SUBAPPLICATION mapping_Uebung_010b3 (* Toggle Flip-Flop mit IE AuxFunction2_X1 *)
  (* Standard: 61499-2; Description: Copyright (c) 2023 Meisterschulen am Ostbahnhof This program and the accompanying materials are made available under the terms of the Eclipse Public License 2.0 which is available at https://www.eclipse.org/legal/epl-2.0/ SPDX-License-Identifier: EPL-2.0 *)
  (* Version 1.0, 2023-10-23, Franz Höpfinger, Meisterschulen am Ostbahnhof *)
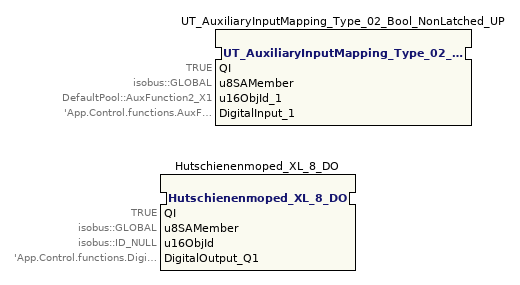
  FBS
    Hutschienenmoped_XL_8_DO : Hutschienenmoped_XL_8_DO(QI := TRUE, u8SAMember := isobus::GLOBAL, u16ObjId := isobus::ID_NULL, DigitalOutput_Q1 := 'App.Control.functions.DigitalOutput_Q1');
    UT_AuxiliaryInputMapping_Type_02_Bool_NonLatched_UP : UT_AuxiliaryInputMapping_Type_02_Bool_NonLatched_UP(QI := TRUE, u8SAMember := isobus::GLOBAL, u16ObjId_1 := DefaultPool::AuxFunction2_X1, DigitalInput_1 := 'App.Control.functions.AuxFunction2_X1');
  END_FBS
END_SUBAPPLICATION
